INTERFACE IEvent_ExecutionAborted EXTENDS IEvent

METHOD RaiseEx
VAR_INPUT
    Message : T_MaxString;
END_VAR
END_METHOD

END_INTERFACE

(* stored: Version 1.1.0.1, ProductVersion 3.1.4024.3
   Itf IEvent_ExecutionAborted: Id {9d5aeb4c-0b5a-055e-0e49-f1cf3b858f36}
   Method RaiseEx: Id {ec680678-cf6f-0159-1239-21001e9fc924} *)
